{attribute 'qualified_only'}
VAR_GLOBAL
	
	System_Start : Int := 1;
	Food_Cut	 : INT  := 0;
	Food_Spiced  : INT  := 0;
	Food_Cooked  : INT  := 0;
	Food_Plated  : INT  := 0;
END_VAR

(* stored: Version 1.1.0.1, ProductVersion 3.1.4024.15
   GVL GVL_Kitchen: Id {babd6c7a-7891-4e66-a650-2261cd14e2f9} *)
